Staubli VAL3: type1.dtx

public TrajSmallBox box{}
